RoboDK station: robotdk_democonveyor.rdk

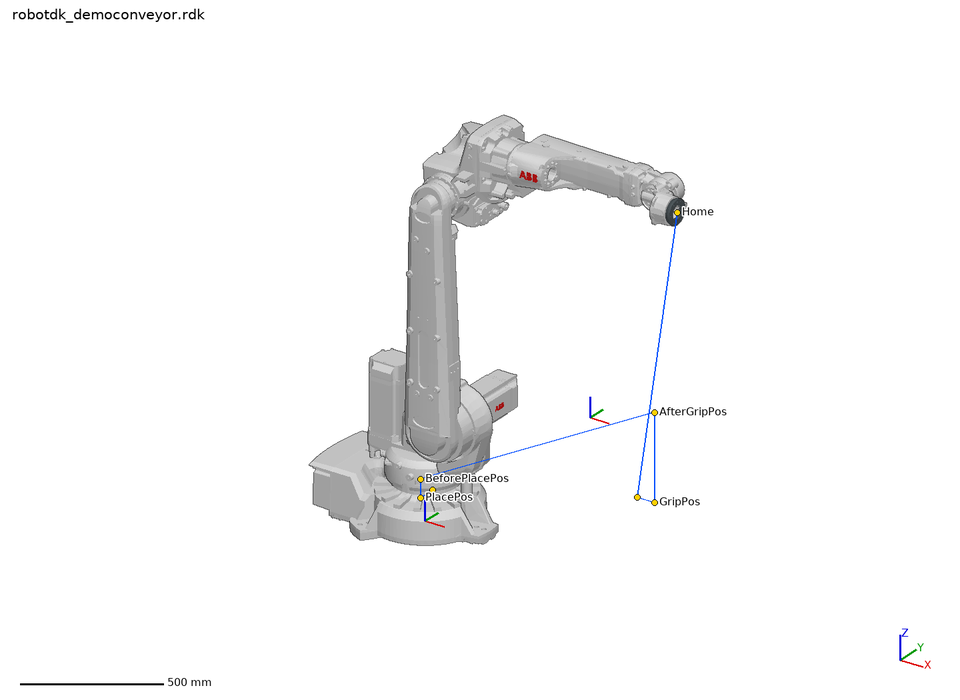
[picture v0: the station drawn from its stored meshes, robots at their saved joint values, targets as dots, program paths as lines]
Station robotdk_democonveyor (saved by RoboDK 5.0.0). Poses are relative to the parent item; angles as X-Y-Z fixed-axis rotations.
Station parameters (name, value as stored): IsAtPick, 0, MoveToPick, 0, IsAtPlace, 0, MoveToPlace, 1, BoxIsPlaced, 0, IO_5, 1
  - frame ABB IRB 2600ID-15/1.85 Base at (0, 0, 0) mm
    - robot ABB IRB 2600ID-15/1.85: 6 axes, payload 15 kg, reach 1850 mm, repeatability 0.026 mm, weight 276 kg
        modified DH rows (alpha deg, a mm, theta deg, d mm): 0, 0, 0, 445; -90, 150, -90, 0; 0, 900, 0, 0; -90, 150, 0, 786; 90, 0, 0, 0; -90, 0, 180, 135
        joint limits [-180, -95, -180, -175, -120, -400] to [180, 155, 75, 175, 120, 400]; home [0, 0, 0, 0, 0, 0]; saved at [0, 0, 0, 0, 0, 0]
    - target Home (Cartesian target) at (1071, 0, 1495) mm, rotated rx 0 ry 90 rz 0 deg; joints [0, 0, 0, 0, 0, 0] of ABB IRB 2600ID-15/1.85
    - target GripPos (Cartesian target) at (1173.89, -282.3, 512.46) mm, rotated rx 0 ry -90 rz -179.34 deg; joints [-15.282, 33.993, 34.831, -17.034, -69.675, 186.074] of ABB IRB 2600ID-15/1.85
    - target AfterGripPos (Cartesian target) at (1173.89, -282.3, 861.45) mm, rotated rx 0 ry -90 rz -179.34 deg; joints [-15.282, 16.906, 27.657, -22.153, -46.759, 195.585] of ABB IRB 2600ID-15/1.85
    - target BeforeGripPos (Cartesian target) at (1099.33, -283.16, 512.46) mm, rotated rx 0 ry -90 rz -179.34 deg; joints [-16.449, 31.408, 40.516, -17.944, -72.75, 185.485] of ABB IRB 2600ID-15/1.85
    - target PlacePos (Cartesian target) at (483.87, -720.12, 512.57) mm, rotated rx 0 ry -90 rz 90 deg; joints [-50.411, 23.299, 59.051, 39.841, -84.112, 175.108] of ABB IRB 2600ID-15/1.85
    - target BeforePlacePos (Cartesian target) at (483.87, -720.12, 585.46) mm, rotated rx 0 ry -90 rz 90 deg; joints [-50.411, 16.895, 58.153, 40.561, -78.532, 170.342] of ABB IRB 2600ID-15/1.85
    - target AfterPlacePos (Cartesian target) at (483.87, -644.96, 512.57) mm, rotated rx 0 ry -90 rz 90 deg; joints [-46.504, 21.636, 63.125, 43.616, -86.202, 176.389] of ABB IRB 2600ID-15/1.85
  - program Prog1 (18 instructions, listed below)
  - frame Frame 2 at (0, 1000, 0) mm
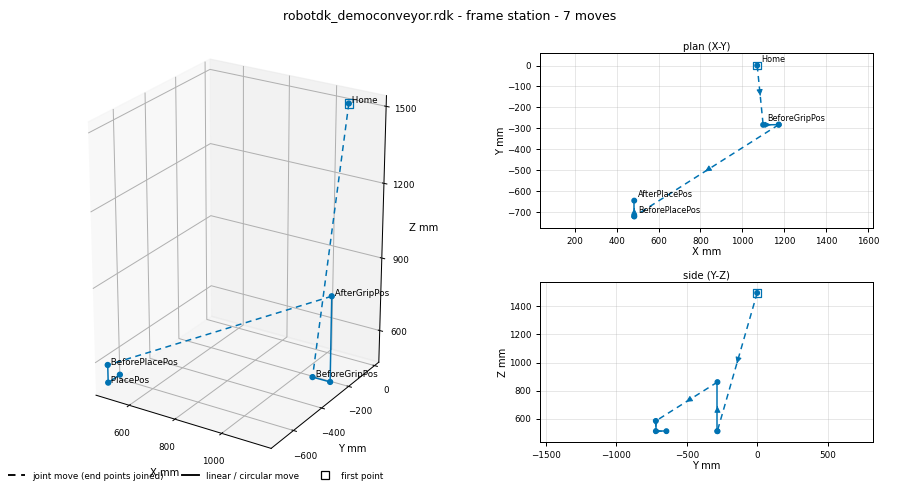
[picture p0: tool path of robotdk_democonveyor.rdk in frame station, 7 of 7 moves have a stored position in this frame; points joined in program order, loops and branches not executed]

--- program Prog1 (robot ABB IRB 2600ID-15/1.85) ---
  Set IsAtPlace=0
  Set IsAtPick=0
  MoveJ (Home)
  Wait MoveToPick=1
  MoveJ (BeforeGripPos)
  Set Ref.: ABB IRB 2600ID-15/1.85 Base
  Set speed (100.0 mm/s)
  MoveL (GripPos)
  Set IsAtPick=1
  Wait MoveToPlace=1
  MoveL (AfterGripPos)
  MoveJ (BeforePlacePos)
  MoveL (PlacePos)
  Set IsAtPlace=1
  Wait BoxIsPlaced=1
  MoveL (AfterPlacePos)
  Set IsAtPlace=0
  Not defined
